{attribute 'qualified_only'}
{attribute 'strict'}
TYPE E_EquipType :
(
	Unknown := 0,
	System := 1,
	Conveyor := 2,
	Merge := 3,
	Gripper_SA := 4,
	Gripper_DA :=5,
	PinStop := 6,
	Pusher := 7,
	Divert := 8
) DINT;
END_TYPE

(* stored: Version 1.1.0.1, ProductVersion 3.1.4024.4
   EnumerationTextList E_EquipType: Id {6dfb7888-8ef8-4b6b-a33f-6300f3e6a13f} *)
